// TIA Portal V15.1 export
// export: Created 2024-05-17T05:38:40.9669861Z, ExportSetting WithDefaults, DisplayName Totally Integrated Automation Portal, DisplayVersion V15.1 Update 5, DisplayName TIA Portal Openness, DisplayVersion V15.1 Update 5, DisplayName SINAMICS Startdrive Advanced, DisplayVersion V15.1, DisplayName G130, G150, S120, S150, SINAMICS MV, S210, DisplayVersion V15.1, DisplayName G110M, G120, G120C, G120D, G120P, DisplayVersion V15.1, DisplayName STEP 7 Professional, DisplayVersion V15.1 Update 5, DisplayName STEP 7 Safety, DisplayVersion V15.1, DisplayName WinCC Professional, DisplayVersion V15.1 Update 5, DisplayName SIMATIC Visualization Architect, DisplayVersion V15.1
FUNCTION "LGBBitShift-Config" : Void   // FC6690, FBD
TITLE = LGBBitShift-Config
{ S7_Optimized_Access := 'TRUE' }
AUTHOR : VCG
VERSION : 0.1
// stored: AutoNumber false, IsIECCheckEnabled false, SetENOAutomatically False, UDAEnableTagReadback false
   VAR_INPUT
      C_Bit0Used : Bool;   // Bit 0 Used
      C_DescriptionBit0 : String;   // Description bit 0
      C_Bit1Used : Bool;   // Bit 1 Used
      C_DescriptionBit1 : String;   // Description bit 1
      C_Bit2Used : Bool;   // Bit 2 Used
      C_DescriptionBit2 : String;   // Description bit 2
      C_Bit3Used : Bool;   // Bit 3 Used
      C_DescriptionBit3 : String;   // Description bit 3
      C_Bit4Used : Bool;   // Bit 4 Used
      C_DescriptionBit4 : String;   // Description bit 4
      C_Bit5Used : Bool;   // Bit 5 Used
      C_DescriptionBit5 : String;   // Description bit 5
      C_Bit6Used : Bool;   // Bit 6 Used
      C_DescriptionBit6 : String;   // Description bit 6
      C_Bit7Used : Bool;   // Bit 7 Used
      C_DescriptionBit7 : String;   // Description bit 7
      C_Bit8Used : Bool;   // Bit 8 Used
      C_DescriptionBit8 : String;   // Description bit 8
      C_Bit9Used : Bool;   // Bit 9 Used
      C_DescriptionBit9 : String;   // Description bit 9
      C_Bit10Used : Bool;   // Bit 10 Used
      C_DescriptionBit10 : String;   // Description bit 10
      C_Bit11Used : Bool;   // Bit 11 Used
      C_DescriptionBit11 : String;   // Description bit 11
      C_Bit12Used : Bool;   // Bit 12 Used
      C_DescriptionBit12 : String;   // Description bit 12
      C_Bit13Used : Bool;   // Bit 13 Used
      C_DescriptionBit13 : String;   // Description bit 13
      C_Bit14Used : Bool;   // Bit 14 Used
      C_DescriptionBit14 : String;   // Description bit 14
      C_Bit15Used : Bool;   // Bit 15 Used
      C_DescriptionBit15 : String;   // Description bit 15
   END_VAR
   VAR_IN_OUT
      IO_Config : "BitShiftConfig";   // Config
   END_VAR
BEGIN

REGION Network 1: **** 1 - Inputs **** Move Config
   // Move Config
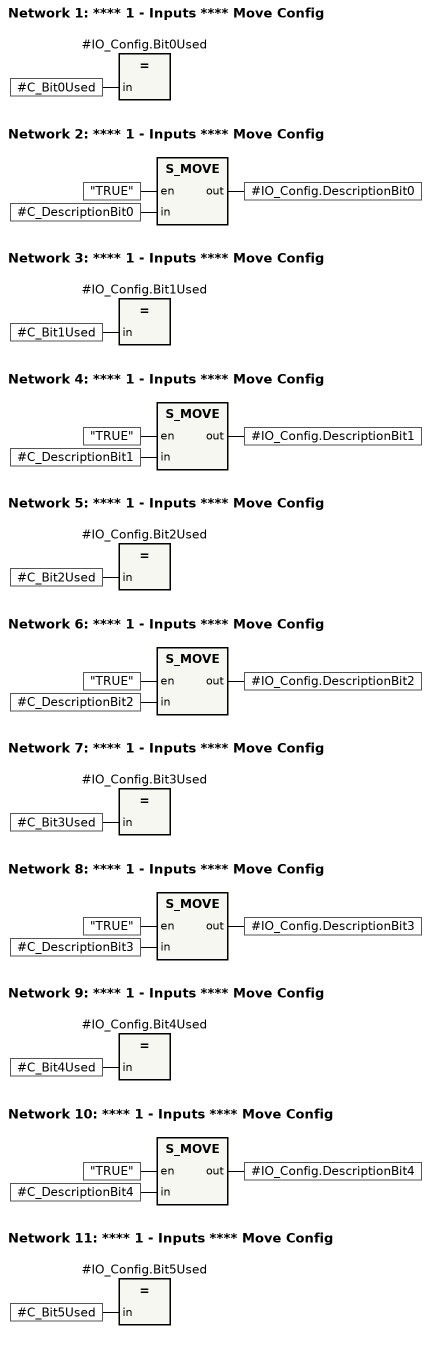
   #IO_Config.Bit0Used := #C_Bit0Used;
END_REGION

REGION Network 2: **** 1 - Inputs **** Move Config
   // Move Config
   IF "TRUE" THEN #IO_Config.DescriptionBit0 := #C_DescriptionBit0; END_IF;
END_REGION

REGION Network 3: **** 1 - Inputs **** Move Config
   // Move Config
   #IO_Config.Bit1Used := #C_Bit1Used;
END_REGION

REGION Network 4: **** 1 - Inputs **** Move Config
   // Move Config
   IF "TRUE" THEN #IO_Config.DescriptionBit1 := #C_DescriptionBit1; END_IF;
END_REGION

REGION Network 5: **** 1 - Inputs **** Move Config
   // Move Config
   #IO_Config.Bit2Used := #C_Bit2Used;
END_REGION

REGION Network 6: **** 1 - Inputs **** Move Config
   // Move Config
   IF "TRUE" THEN #IO_Config.DescriptionBit2 := #C_DescriptionBit2; END_IF;
END_REGION

REGION Network 7: **** 1 - Inputs **** Move Config
   // Move Config
   #IO_Config.Bit3Used := #C_Bit3Used;
END_REGION

REGION Network 8: **** 1 - Inputs **** Move Config
   // Move Config
   IF "TRUE" THEN #IO_Config.DescriptionBit3 := #C_DescriptionBit3; END_IF;
END_REGION

REGION Network 9: **** 1 - Inputs **** Move Config
   // Move Config
   #IO_Config.Bit4Used := #C_Bit4Used;
END_REGION

REGION Network 10: **** 1 - Inputs **** Move Config
   // Move Config
   IF "TRUE" THEN #IO_Config.DescriptionBit4 := #C_DescriptionBit4; END_IF;
END_REGION

REGION Network 11: **** 1 - Inputs **** Move Config
   // Move Config
   #IO_Config.Bit5Used := #C_Bit5Used;
END_REGION

REGION Network 12: **** 1 - Inputs **** Move Config
   // Move Config
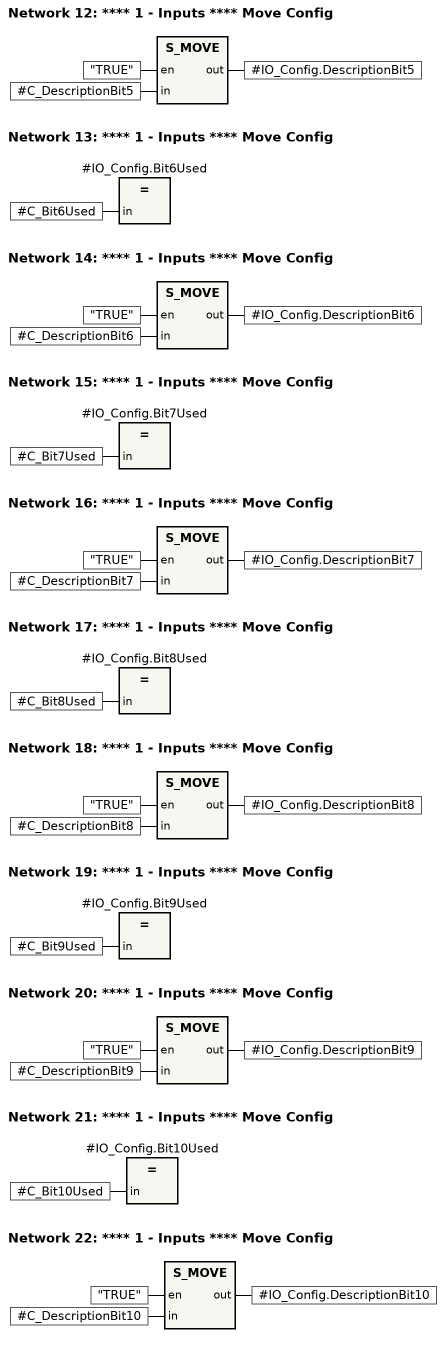
   IF "TRUE" THEN #IO_Config.DescriptionBit5 := #C_DescriptionBit5; END_IF;
END_REGION

REGION Network 13: **** 1 - Inputs **** Move Config
   // Move Config
   #IO_Config.Bit6Used := #C_Bit6Used;
END_REGION

REGION Network 14: **** 1 - Inputs **** Move Config
   // Move Config
   IF "TRUE" THEN #IO_Config.DescriptionBit6 := #C_DescriptionBit6; END_IF;
END_REGION

REGION Network 15: **** 1 - Inputs **** Move Config
   // Move Config
   #IO_Config.Bit7Used := #C_Bit7Used;
END_REGION

REGION Network 16: **** 1 - Inputs **** Move Config
   // Move Config
   IF "TRUE" THEN #IO_Config.DescriptionBit7 := #C_DescriptionBit7; END_IF;
END_REGION

REGION Network 17: **** 1 - Inputs **** Move Config
   // Move Config
   #IO_Config.Bit8Used := #C_Bit8Used;
END_REGION

REGION Network 18: **** 1 - Inputs **** Move Config
   // Move Config
   IF "TRUE" THEN #IO_Config.DescriptionBit8 := #C_DescriptionBit8; END_IF;
END_REGION

REGION Network 19: **** 1 - Inputs **** Move Config
   // Move Config
   #IO_Config.Bit9Used := #C_Bit9Used;
END_REGION

REGION Network 20: **** 1 - Inputs **** Move Config
   // Move Config
   IF "TRUE" THEN #IO_Config.DescriptionBit9 := #C_DescriptionBit9; END_IF;
END_REGION

REGION Network 21: **** 1 - Inputs **** Move Config
   // Move Config
   #IO_Config.Bit10Used := #C_Bit10Used;
END_REGION

REGION Network 22: **** 1 - Inputs **** Move Config
   // Move Config
   IF "TRUE" THEN #IO_Config.DescriptionBit10 := #C_DescriptionBit10; END_IF;
END_REGION

REGION Network 23: **** 1 - Inputs **** Move Config
   // Move Config
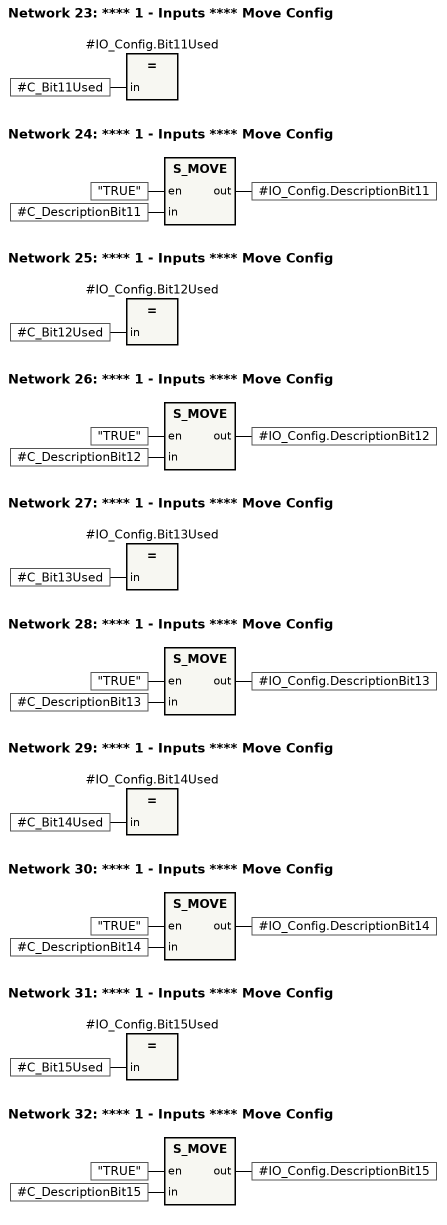
   #IO_Config.Bit11Used := #C_Bit11Used;
END_REGION

REGION Network 24: **** 1 - Inputs **** Move Config
   // Move Config
   IF "TRUE" THEN #IO_Config.DescriptionBit11 := #C_DescriptionBit11; END_IF;
END_REGION

REGION Network 25: **** 1 - Inputs **** Move Config
   // Move Config
   #IO_Config.Bit12Used := #C_Bit12Used;
END_REGION

REGION Network 26: **** 1 - Inputs **** Move Config
   // Move Config
   IF "TRUE" THEN #IO_Config.DescriptionBit12 := #C_DescriptionBit12; END_IF;
END_REGION

REGION Network 27: **** 1 - Inputs **** Move Config
   // Move Config
   #IO_Config.Bit13Used := #C_Bit13Used;
END_REGION

REGION Network 28: **** 1 - Inputs **** Move Config
   // Move Config
   IF "TRUE" THEN #IO_Config.DescriptionBit13 := #C_DescriptionBit13; END_IF;
END_REGION

REGION Network 29: **** 1 - Inputs **** Move Config
   // Move Config
   #IO_Config.Bit14Used := #C_Bit14Used;
END_REGION

REGION Network 30: **** 1 - Inputs **** Move Config
   // Move Config
   IF "TRUE" THEN #IO_Config.DescriptionBit14 := #C_DescriptionBit14; END_IF;
END_REGION

REGION Network 31: **** 1 - Inputs **** Move Config
   // Move Config
   #IO_Config.Bit15Used := #C_Bit15Used;
END_REGION

REGION Network 32: **** 1 - Inputs **** Move Config
   // Move Config
   IF "TRUE" THEN #IO_Config.DescriptionBit15 := #C_DescriptionBit15; END_IF;
END_REGION
END_FUNCTION
